// TIA Portal V17 export
// export: Created 2022-07-20T06:59:47.6094645Z, ExportSetting WithDefaults, DisplayName Totally Integrated Automation Portal, DisplayVersion V17, DisplayName TIA Portal Openness, DisplayVersion V17, DisplayName TIA Portal Version Control Interface, DisplayVersion V17, DisplayName SINAMICS Startdrive Advanced, DisplayVersion V17, DisplayName SINAMICS Startdrive G130, G150, S120, S150, SINAMICS MV, S210, DisplayVersion V17, DisplayName SINAMICS Startdrive G110M, G120, G120C, G120D, G120P, G115D, DisplayVersion V17, DisplayName STEP 7 Professional, DisplayVersion V17, DisplayName STEP 7 Safety, DisplayVersion V17, DisplayName WinCC Advanced, DisplayVersion V17
FUNCTION_BLOCK "FB10150_MDPModbusStepperMotorManager"   // FB10150, LAD
TITLE = FB10150_MDPModbusStepperMotorManager
{ S7_Optimized_Access := 'TRUE' }
AUTHOR : Anirouddh
FAMILY : 1015x_MDP
VERSION : 1.0
// Release note : 
// 1.0 - Feature developped
// stored: AutoNumber false, IsIECCheckEnabled false, IsRetainMemResEnabled false, MemoryReserve 100, SetENOAutomatically false, UDAEnableTagReadback false
   VAR_INPUT
      MotorInError : Bool;
      OriginPosition : Real;
      WorkingPosition : Real;
      StepsMmRatio : Real;
      RequestAcknowledge : Bool;
      RequestHoming : Bool;
      RequestExecuteQProgram : Bool;
      RequestGoToOriginPosition : Bool;
      RequestGoToWorkingPosition : Bool;
      RequestWriteOriginPosition : Bool;
      RequestWriteWorkingPosition : Bool;
      RequestReadActualPosition : Bool;
      RequestReadOriginPosition : Bool;
      RequestReadWorkingPosition : Bool;
      ModbusRequestDone : Bool;
      ModbusDataRegisterToReceive_0 : Int;
      ModbusDataRegisterToReceive_1 : Int;
   END_VAR
   VAR_OUTPUT
      StartMovement : Bool;
      DoHoming : Bool;
      GoToWorkingPosition : Bool;
      AlarmReset : Bool;
      ActualPosition : Real;
      ActualOriginPosition : Real;
      ActualWorkingPosition : Real;
      HomingDone : Bool;
      IsInOriginPosition : Bool;
      IsInWorkingPosition : Bool;
      ReadActualPositionDone : Bool;
      ReadOriginPositionDone : Bool;
      ReadWorkingPositionDone : Bool;
      ReadAlarmStatusDone : Bool;
      WriteOriginPositionDone : Bool;
      WriteWorkingPositionDone : Bool;
      StartModbusRtuCommunication : Bool;
      ModbusRtuDataAddress : UInt;
      ModbusRtuDataLength : UInt;
      ModbusRtuMode : USInt;
      ModbusDataRegisterToSend_0 : Int;
      ModbusDataRegisterToSend_1 : Int;
      AlarmStatus : Int;
      MaterialOK : Bool;
   END_VAR
   VAR
      RequestMotorStartUp : Bool;
      MotorStartUpStateDiagram : Int;
      ModbusCommunicationStateDiagram : Int;
      MotorMovementStateDiagram : Int;
      MotorAlarmManagementStateDiagram : Int;
      R_TRIG_RequestHoming { S7_SetPoint := 'True'} : R_TRIG;
      R_TRIG_RequestGoToOriginPosition { S7_SetPoint := 'True'} : R_TRIG;
      R_TRIG_RequestGoToWorkingPosition { S7_SetPoint := 'True'} : R_TRIG;
      R_TRIG_ModbusRequestDone { S7_SetPoint := 'True'} : R_TRIG;
      R_TRIG_RequestAcknowledge { S7_SetPoint := 'True'} : R_TRIG;
      F_TRIG_MotorInError { S7_SetPoint := 'True'} : R_TRIG;
      TON_HomingSignal { S7_SetPoint := 'True'} : TON_TIME;
      TON_GoToWorkingPositionSignal { S7_SetPoint := 'True'} : TON_TIME;
      TON_GoToOriginPositionSignal { S7_SetPoint := 'True'} : TON_TIME;
      TON_AlarmResetSignal { S7_SetPoint := 'True'} : TON_TIME;
   END_VAR
   VAR_TEMP
      ActualPositionTemp : DInt;
      ActualOriginPositionTemp : DInt;
      ActualWorkingPositionTemp : DInt;
      BlankAlarmCode : Array[0..15] of Bool;
   END_VAR
   VAR CONSTANT
      WAIT_FOR_MOTOR_START_UP : Int := 0;
      EXECUTE_Q_PROGRAM : Int := 10;
      INITIALIZE_ORIGIN_POSITION : Int := 20;
      INITIALIZE_WORKING_POSITION : Int := 30;
      MOTOR_START_UP_DONE : Int := 40;
      "==========" : Bool;
      WAIT_FOR_MODBUS_COMMUNICATION_REQUEST : Int := 0;
      READ_ACTUAL_POSITION : Int := 10;
      READ_ORIGIN_POSITION : Int := 20;
      READ_WORKING_POSITION : Int := 30;
      WRITE_ORIGIN_POSITION : Int := 40;
      WRITE_WORKING_POSITION : Int := 50;
      MODBUS_COMMUNICATION_DONE : Int := 70;
      "==========_1" : Bool;
      WAIT_FOR_MOVEMENT_REQUEST : Int := 0;
      HOMING : Int := 10;
      GO_TO_ORIGIN_POSITION : Int := 20;
      GO_TO_WORKING_POSITION : Int := 30;
      MOVEMENT_DONE : Int := 40;
      "==========_2" : Bool;
      WAIT_FOR_MOTOR_ERROR : Int := 0;
      RESET_MOTOR_COMMUNICATION_MOVEMENT : Int := 10;
      ALARM_RESET : Int := 20;
      GATHER_ERROR_CODE : Int := 30;
      MOTOR_ERROR_MANAGEMENT_DONE : Int := 40;
   END_VAR
BEGIN

REGION Network 1 (SCL): First Scan
   IF "FirstScan" THEN
       #RequestMotorStartUp := TRUE;
       #MaterialOK := FALSE;
       #HomingDone := FALSE;
       #IsInOriginPosition := FALSE;
       #IsInWorkingPosition := FALSE;
       #ReadActualPositionDone := FALSE; 
       #ReadOriginPositionDone := FALSE;
       #ReadWorkingPositionDone := FALSE;
       #WriteOriginPositionDone := FALSE;
       #WriteWorkingPositionDone := FALSE;
       #StartMovement := FALSE;
       #DoHoming := FALSE;
       #GoToWorkingPosition := FALSE;
       #MotorStartUpStateDiagram := #WAIT_FOR_MOTOR_START_UP;
       #ModbusCommunicationStateDiagram := #WAIT_FOR_MODBUS_COMMUNICATION_REQUEST;
       #MotorMovementStateDiagram := #WAIT_FOR_MOVEMENT_REQUEST;
   END_IF;
END_REGION

REGION Network 2 (SCL): Motor Start Up Sequence
   CASE #MotorStartUpStateDiagram OF
       #WAIT_FOR_MOTOR_START_UP:
           IF #RequestMotorStartUp AND #RequestAcknowledge THEN
               #MotorStartUpStateDiagram := #EXECUTE_Q_PROGRAM;
           END_IF;
       #EXECUTE_Q_PROGRAM:
           #StartModbusRtuCommunication := TRUE;
           #ModbusRtuDataAddress := 40126;
           #ModbusRtuDataLength := 1;
           #ModbusRtuMode := "MODBUS_RTU_WRITE_MODE";
           #ModbusDataRegisterToSend_0 := 1;
           #R_TRIG_ModbusRequestDone(CLK := #ModbusRequestDone);
           IF #R_TRIG_ModbusRequestDone.Q THEN
               #StartModbusRtuCommunication := FALSE;
               #MotorStartUpStateDiagram := #INITIALIZE_ORIGIN_POSITION;
           END_IF;
       #INITIALIZE_ORIGIN_POSITION:
           #StartModbusRtuCommunication := TRUE;
           #ModbusRtuDataAddress := 40061;
           #ModbusRtuDataLength := 2;
           #ModbusRtuMode := "MODBUS_RTU_WRITE_MODE";
           "FC10332_DWordTo2Words"(DWord_Input := REAL_TO_DINT(#OriginPosition * #StepsMmRatio),
                                Word_HighWeight => #ModbusDataRegisterToSend_0,
                                Word_LowWeight => #ModbusDataRegisterToSend_1);
           #R_TRIG_ModbusRequestDone(CLK := #ModbusRequestDone);
           IF #R_TRIG_ModbusRequestDone.Q THEN
               #WriteOriginPositionDone := TRUE;
               #StartModbusRtuCommunication := FALSE;
               #MotorStartUpStateDiagram := #INITIALIZE_WORKING_POSITION;
           END_IF;
       #INITIALIZE_WORKING_POSITION:
           #StartModbusRtuCommunication := TRUE;
           #ModbusRtuDataAddress := 40063;
           #ModbusRtuDataLength := 2;
           #ModbusRtuMode := "MODBUS_RTU_WRITE_MODE";
           "FC10332_DWordTo2Words"(DWord_Input := REAL_TO_DINT(#WorkingPosition * #StepsMmRatio),
                                Word_HighWeight => #ModbusDataRegisterToSend_0,
                                Word_LowWeight => #ModbusDataRegisterToSend_1);
           #R_TRIG_ModbusRequestDone(CLK := #ModbusRequestDone);
           IF #R_TRIG_ModbusRequestDone.Q THEN
               #WriteWorkingPositionDone := TRUE;
               #StartModbusRtuCommunication := FALSE;
               #MotorStartUpStateDiagram := #MOTOR_START_UP_DONE;
           END_IF;
       #MOTOR_START_UP_DONE:
           #MaterialOK := TRUE;
           #RequestMotorStartUp := FALSE;
   END_CASE;
END_REGION

REGION Network 3 (SCL): Modbus Communication Management
   CASE #ModbusCommunicationStateDiagram OF
       #WAIT_FOR_MODBUS_COMMUNICATION_REQUEST:
           IF #RequestReadActualPosition (* OR (#HomingDone AND "Clock_0.5Hz") *)THEN
               #ReadOriginPositionDone := FALSE;
               #ReadWorkingPositionDone := FALSE;
               #ReadActualPositionDone := FALSE;
               #WriteOriginPositionDone := FALSE;
               #WriteWorkingPositionDone := FALSE;
               #ModbusCommunicationStateDiagram := #READ_ACTUAL_POSITION;
           ELSIF #RequestReadOriginPosition THEN
               #ReadOriginPositionDone := FALSE;
               #ReadWorkingPositionDone := FALSE;
               #ReadActualPositionDone := FALSE;
               #WriteOriginPositionDone := FALSE;
               #WriteWorkingPositionDone := FALSE;
               #ModbusCommunicationStateDiagram := #READ_ORIGIN_POSITION;
           ELSIF #RequestReadWorkingPosition THEN
               #ReadOriginPositionDone := FALSE;
               #ReadWorkingPositionDone := FALSE;
               #ReadActualPositionDone := FALSE;
               #WriteOriginPositionDone := FALSE;
               #WriteWorkingPositionDone := FALSE;
               #ModbusCommunicationStateDiagram := #READ_WORKING_POSITION;
           ELSIF #RequestWriteOriginPosition THEN
               #ReadOriginPositionDone := FALSE;
               #ReadWorkingPositionDone := FALSE;
               #ReadActualPositionDone := FALSE;
               #WriteOriginPositionDone := FALSE;
               #WriteWorkingPositionDone := FALSE;
               #ReadActualPositionDone := FALSE;
               #ModbusCommunicationStateDiagram := #WRITE_ORIGIN_POSITION;
           ELSIF #RequestWriteWorkingPosition THEN
               #ReadOriginPositionDone := FALSE;
               #ReadWorkingPositionDone := FALSE;
               #ReadActualPositionDone := FALSE;
               #WriteOriginPositionDone := FALSE;
               #WriteWorkingPositionDone := FALSE;
               #ModbusCommunicationStateDiagram := #WRITE_WORKING_POSITION;
           ELSIF "FirstScan" OR #RequestExecuteQProgram THEN
               #ModbusCommunicationStateDiagram := #EXECUTE_Q_PROGRAM;
           END_IF;
       #READ_ACTUAL_POSITION:
           #StartModbusRtuCommunication := TRUE;
           #ModbusRtuDataAddress := 40007;
           #ModbusRtuDataLength := 2;
           #ModbusRtuMode := "MODBUS_RTU_READ_MODE";
           IF #ModbusRequestDone THEN
               "FC10012_2IntToDint"(HighInt := #ModbusDataRegisterToReceive_0,
                                    LowInt := #ModbusDataRegisterToReceive_1,
                                    Output_DInt => #ActualPositionTemp);
               #ActualPosition := DINT_TO_REAL(#ActualPositionTemp) /#StepsMmRatio;
               #ReadActualPositionDone := TRUE;
               #StartModbusRtuCommunication := FALSE;
               #ModbusCommunicationStateDiagram := #MODBUS_COMMUNICATION_DONE;
           END_IF;
       #READ_ORIGIN_POSITION:
           #StartModbusRtuCommunication := TRUE;
           #ModbusRtuDataAddress := 40061;
           #ModbusRtuDataLength := 2;
           #ModbusRtuMode := "MODBUS_RTU_READ_MODE";
           IF #ModbusRequestDone THEN
               "FC10012_2IntToDint"(HighInt := #ModbusDataRegisterToReceive_0,
                                    LowInt := #ModbusDataRegisterToReceive_1,
                                    Output_DInt => #ActualOriginPositionTemp);
               #ActualOriginPosition := DINT_TO_REAL(#ActualOriginPositionTemp) / #StepsMmRatio;
               #ReadOriginPositionDone := TRUE;
               #StartModbusRtuCommunication := FALSE;
               #ModbusCommunicationStateDiagram := #MODBUS_COMMUNICATION_DONE;
           END_IF;
       #READ_WORKING_POSITION:
           #StartModbusRtuCommunication := TRUE;
           #ModbusRtuDataAddress := 40063;
           #ModbusRtuDataLength := 2;
           #ModbusRtuMode := "MODBUS_RTU_READ_MODE";
           IF #ModbusRequestDone THEN
               "FC10012_2IntToDint"(HighInt := #ModbusDataRegisterToReceive_0,
                                    LowInt := #ModbusDataRegisterToReceive_1,
                                    Output_DInt => #ActualWorkingPositionTemp);
               #ActualWorkingPosition := DINT_TO_REAL(#ActualWorkingPositionTemp) / #StepsMmRatio;
               #ReadWorkingPositionDone := TRUE;
               #StartModbusRtuCommunication := FALSE;
               #ModbusCommunicationStateDiagram := #MODBUS_COMMUNICATION_DONE;
           END_IF;
       #WRITE_ORIGIN_POSITION:
           #StartModbusRtuCommunication := TRUE;
           #ModbusRtuDataAddress := 40061;
           #ModbusRtuDataLength := 2;
           #ModbusRtuMode := "MODBUS_RTU_WRITE_MODE";
           "FC10332_DWordTo2Words"(DWord_Input := REAL_TO_DINT(#OriginPosition * #StepsMmRatio),
                                Word_HighWeight => #ModbusDataRegisterToSend_0,
                                Word_LowWeight => #ModbusDataRegisterToSend_1);
           IF #ModbusRequestDone THEN
               #WriteOriginPositionDone := TRUE;
               #StartModbusRtuCommunication := FALSE;
               #ModbusCommunicationStateDiagram := #MODBUS_COMMUNICATION_DONE;
           END_IF;
       #WRITE_WORKING_POSITION:
           #StartModbusRtuCommunication := TRUE;
           #ModbusRtuDataAddress := 40063;
           #ModbusRtuDataLength := 2;
           #ModbusRtuMode := "MODBUS_RTU_WRITE_MODE";
           "FC10332_DWordTo2Words"(DWord_Input := REAL_TO_DINT(#WorkingPosition * #StepsMmRatio),
                                Word_HighWeight => #ModbusDataRegisterToSend_0,
                                Word_LowWeight => #ModbusDataRegisterToSend_1);
           IF #ModbusRequestDone THEN
               #WriteWorkingPositionDone := TRUE;
               #StartModbusRtuCommunication := FALSE;
               #ModbusCommunicationStateDiagram := #MODBUS_COMMUNICATION_DONE;
           END_IF;
       #MODBUS_COMMUNICATION_DONE:
           #ModbusCommunicationStateDiagram := #WAIT_FOR_MODBUS_COMMUNICATION_REQUEST;
   END_CASE;
END_REGION

REGION Network 4 (SCL): Motor Movement Management
   CASE #MotorMovementStateDiagram OF
       #WAIT_FOR_MOVEMENT_REQUEST:
           #R_TRIG_RequestHoming(CLK := #RequestHoming);
           #R_TRIG_RequestGoToOriginPosition(CLK := #RequestGoToOriginPosition);
           #R_TRIG_RequestGoToWorkingPosition(CLK := #RequestGoToWorkingPosition);
           IF #R_TRIG_RequestGoToOriginPosition.Q THEN
               #HomingDone := FALSE;
               #IsInOriginPosition := FALSE;
               #IsInWorkingPosition := FALSE;
               #MotorMovementStateDiagram := #GO_TO_ORIGIN_POSITION;
           ELSIF #R_TRIG_RequestGoToWorkingPosition.Q THEN
               #HomingDone := FALSE;
               #IsInOriginPosition := FALSE;
               #IsInWorkingPosition := FALSE;
               #MotorMovementStateDiagram := #GO_TO_WORKING_POSITION;
           ELSIF #R_TRIG_RequestHoming.Q THEN
               #HomingDone := FALSE;
               #IsInOriginPosition := FALSE;
               #IsInWorkingPosition := FALSE;
               #MotorMovementStateDiagram := #HOMING;
           END_IF;
       #HOMING:
           #DoHoming := TRUE;
           #HomingDone := FALSE;
           IF #TON_HomingSignal.Q THEN
               #DoHoming := FALSE;
               #HomingDone := TRUE;
               #MotorMovementStateDiagram := #MOVEMENT_DONE;
           END_IF;
       #GO_TO_ORIGIN_POSITION:
           #StartMovement := TRUE;
           #GoToWorkingPosition := FALSE;
           IF #TON_GoToOriginPositionSignal.Q THEN
               #IsInOriginPosition := TRUE;
               #StartMovement := FALSE;
               #GoToWorkingPosition := FALSE;
               #MotorMovementStateDiagram := #MOVEMENT_DONE;
           END_IF;
       #GO_TO_WORKING_POSITION:
           #StartMovement := TRUE;
           #GoToWorkingPosition := TRUE;
           IF #TON_GoToWorkingPositionSignal.Q THEN
               #IsInWorkingPosition := TRUE;
               #StartMovement := FALSE;
               #GoToWorkingPosition := FALSE;
               #MotorMovementStateDiagram := #MOVEMENT_DONE;
           END_IF;
       #MOVEMENT_DONE:
           #MotorMovementStateDiagram := #WAIT_FOR_MOVEMENT_REQUEST;
   END_CASE;
END_REGION

REGION Network 5 (SCL): Motor Error Management
   CASE #MotorAlarmManagementStateDiagram OF
       #WAIT_FOR_MOTOR_ERROR:
           #F_TRIG_MotorInError(CLK := #MotorInError);
           #R_TRIG_RequestAcknowledge(CLK := #RequestAcknowledge);
           IF #F_TRIG_MotorInError.Q THEN
               #ReadAlarmStatusDone := FALSE;
               #MotorAlarmManagementStateDiagram := #RESET_MOTOR_COMMUNICATION_MOVEMENT;
           ELSIF #R_TRIG_RequestAcknowledge.Q THEN
               #ReadAlarmStatusDone := FALSE;
               #MotorAlarmManagementStateDiagram := #ALARM_RESET;
           END_IF;
       #RESET_MOTOR_COMMUNICATION_MOVEMENT:
           #ModbusCommunicationStateDiagram := #WAIT_FOR_MODBUS_COMMUNICATION_REQUEST;
           #MotorMovementStateDiagram := #WAIT_FOR_MOVEMENT_REQUEST;
           #StartMovement := FALSE;
           #GoToWorkingPosition := FALSE;
           #DoHoming := FALSE;
           #StartModbusRtuCommunication := FALSE;
           IF #ModbusCommunicationStateDiagram = #WAIT_FOR_MODBUS_COMMUNICATION_REQUEST AND #MotorMovementStateDiagram = #WAIT_FOR_MOVEMENT_REQUEST AND NOT(#StartModbusRtuCommunication) THEN
               #MotorAlarmManagementStateDiagram := #GATHER_ERROR_CODE;
           END_IF;
       #ALARM_RESET:
           #AlarmReset := TRUE;
           IF #TON_AlarmResetSignal.Q THEN
               #AlarmReset := FALSE;
               #MotorAlarmManagementStateDiagram := #GATHER_ERROR_CODE;
           END_IF;
       #GATHER_ERROR_CODE:
           #StartModbusRtuCommunication := TRUE;
           #ModbusRtuDataAddress := 40001;
           #ModbusRtuDataLength := 1;
           #ModbusRtuMode := "MODBUS_RTU_READ_MODE";
           IF #ModbusRequestDone THEN
               #AlarmStatus := #ModbusDataRegisterToSend_0;
               #ReadAlarmStatusDone := TRUE;
               #AlarmReset := FALSE;
               #StartModbusRtuCommunication := FALSE;
               #MotorAlarmManagementStateDiagram := #MOTOR_ERROR_MANAGEMENT_DONE;
           END_IF;
       #MOTOR_ERROR_MANAGEMENT_DONE:
           #MotorAlarmManagementStateDiagram := #WAIT_FOR_MOTOR_ERROR;
   END_CASE;
END_REGION

REGION Network 6 (SCL): Signal Timers
   //HomingSignal
   #TON_HomingSignal(IN := #DoHoming,
                     PT := T#500ms);

   //GoToWorkingPositionSignal
   #TON_GoToWorkingPositionSignal(IN := #StartMovement AND #GoToWorkingPosition,
                                  PT := T#1s);

   //GoToOriginPositionSiganl
   #TON_GoToOriginPositionSignal(IN := #StartMovement AND NOT(#GoToWorkingPosition),
                                 PT := T#1s);

   //AcknowledgeSignal
   #TON_AlarmResetSignal(IN := #MotorAlarmManagementStateDiagram = #ALARM_RESET,
                          PT := T#300ms);
END_REGION
END_FUNCTION_BLOCK
